// TIA Portal V18 export
// export: Created 2026-01-09T11:32:01.0889439Z, ExportSetting WithDefaults, DisplayName Totally Integrated Automation Portal, DisplayVersion V18 Update 5, DisplayName TIA Portal Openness, DisplayVersion V18 Update 5, DisplayName TIA Portal Teamcenter Gateway, DisplayVersion V18, DisplayName TIA Portal Version Control Interface, DisplayVersion V18, DisplayName SINAMICS Startdrive Advanced, DisplayVersion V18 SP2 Update 1, DisplayName SINAMICS Startdrive G110M, G120, G120C, G120D, G120P, G115D, DisplayVersion V18 SP2 Update 1, DisplayName SINAMICS Startdrive G130, G150, S120, S150, SINAMICS MV, S210, G220, S200, DisplayVersion V18 SP2 Update 1, DisplayName STEP 7 Professional, DisplayVersion V18 Update 5, DisplayName STEP 7 Safety, DisplayVersion V18, DisplayName WinCC Professional, DisplayVersion V18 Update 5
TagTable "Pilz"
  PilzData_85A1_I8 : Bool  (PLC tag PilzData.85A1.I8, CPU S71500-2PN_TP700, 100 ms)
  PilzData_85A1_I9 : Bool  (PLC tag PilzData.85A1.I9, CPU S71500-2PN_TP700, 100 ms)
  PilzData_85A1_I10 : Bool  (PLC tag PilzData.85A1.I10, CPU S71500-2PN_TP700, 100 ms)
  PilzData_85A1_I11 : Bool  (PLC tag PilzData.85A1.I11, CPU S71500-2PN_TP700, 100 ms)
  PilzData_85A1_I12 : Bool  (PLC tag PilzData.85A1.I12, CPU S71500-2PN_TP700, 100 ms)
  PilzData_85A1_I13 : Bool  (PLC tag PilzData.85A1.I13, CPU S71500-2PN_TP700, 100 ms)
  PilzData_85A1_I14 : Bool  (PLC tag PilzData.85A1.I14, CPU S71500-2PN_TP700, 100 ms)
  PilzData_85A1_I15 : Bool  (PLC tag PilzData.85A1.I15, CPU S71500-2PN_TP700, 100 ms)
  PilzData_85A1_I0 : Bool  (PLC tag PilzData.85A1.I0, CPU S71500-2PN_TP700, 100 ms)
  PilzData_85A1_I1 : Bool  (PLC tag PilzData.85A1.I1, CPU S71500-2PN_TP700, 100 ms)
  PilzData_85A1_I2 : Bool  (PLC tag PilzData.85A1.I2, CPU S71500-2PN_TP700, 100 ms)
  PilzData_85A1_I3 : Bool  (PLC tag PilzData.85A1.I3, CPU S71500-2PN_TP700, 100 ms)
  PilzData_85A1_I4 : Bool  (PLC tag PilzData.85A1.I4, CPU S71500-2PN_TP700, 100 ms)
  PilzData_85A1_I5 : Bool  (PLC tag PilzData.85A1.I5, CPU S71500-2PN_TP700, 100 ms)
  PilzData_85A1_I6 : Bool  (PLC tag PilzData.85A1.I6, CPU S71500-2PN_TP700, 100 ms)
  PilzData_85A1_I7 : Bool  (PLC tag PilzData.85A1.I7, CPU S71500-2PN_TP700, 100 ms)
  PilzData_85A1_I24 : Bool  (PLC tag PilzData.85A1.I24, CPU S71500-2PN_TP700, 100 ms)
  PilzData_85A1_I25 : Bool  (PLC tag PilzData.85A1.I25, CPU S71500-2PN_TP700, 100 ms)
  PilzData_85A1_I26 : Bool  (PLC tag PilzData.85A1.I26, CPU S71500-2PN_TP700, 100 ms)
  PilzData_85A1_I27 : Bool  (PLC tag PilzData.85A1.I27, CPU S71500-2PN_TP700, 100 ms)
  PilzData_85A1_I28 : Bool  (PLC tag PilzData.85A1.I28, CPU S71500-2PN_TP700, 100 ms)
  PilzData_85A1_I29 : Bool  (PLC tag PilzData.85A1.I29, CPU S71500-2PN_TP700, 100 ms)
  PilzData_85A1_I30 : Bool  (PLC tag PilzData.85A1.I30, CPU S71500-2PN_TP700, 100 ms)
  PilzData_85A1_I31 : Bool  (PLC tag PilzData.85A1.I31, CPU S71500-2PN_TP700, 100 ms)
  PilzData_85A1_I16 : Bool  (PLC tag PilzData.85A1.I16, CPU S71500-2PN_TP700, 100 ms)
  PilzData_85A1_I17 : Bool  (PLC tag PilzData.85A1.I17, CPU S71500-2PN_TP700, 100 ms)
  PilzData_85A1_I18 : Bool  (PLC tag PilzData.85A1.I18, CPU S71500-2PN_TP700, 100 ms)
  PilzData_85A1_I19 : Bool  (PLC tag PilzData.85A1.I19, CPU S71500-2PN_TP700, 100 ms)
  PilzData_85A1_I20 : Bool  (PLC tag PilzData.85A1.I20, CPU S71500-2PN_TP700, 100 ms)
  PilzData_85A1_I21 : Bool  (PLC tag PilzData.85A1.I21, CPU S71500-2PN_TP700, 100 ms)
  PilzData_85A1_I22 : Bool  (PLC tag PilzData.85A1.I22, CPU S71500-2PN_TP700, 100 ms)
  PilzData_85A1_I23 : Bool  (PLC tag PilzData.85A1.I23, CPU S71500-2PN_TP700, 100 ms)
  PilzData_85A1_O0 : Bool  (PLC tag PilzData.85A1.O0, CPU S71500-2PN_TP700, 100 ms)
  PilzData_85A1_O1 : Bool  (PLC tag PilzData.85A1.O1, CPU S71500-2PN_TP700, 100 ms)
  PilzData_85A1_O2 : Bool  (PLC tag PilzData.85A1.O2, CPU S71500-2PN_TP700, 100 ms)
  PilzData_85A1_O3 : Bool  (PLC tag PilzData.85A1.O3, CPU S71500-2PN_TP700, 100 ms)
  PilzData_85A1_Spare_1 : Bool  (PLC tag PilzData.85A1.Spare_1, CPU S71500-2PN_TP700, 100 ms)
  PilzData_85A1_Spare_2 : Bool  (PLC tag PilzData.85A1.Spare_2, CPU S71500-2PN_TP700, 100 ms)
  PilzData_85A1_Spare_3 : Bool  (PLC tag PilzData.85A1.Spare_3, CPU S71500-2PN_TP700, 100 ms)
  PilzData_85A1_Spare_4 : Bool  (PLC tag PilzData.85A1.Spare_4, CPU S71500-2PN_TP700, 100 ms)
  PilzData_85A1_Spare_5 : Bool  (PLC tag PilzData.85A1.Spare_5, CPU S71500-2PN_TP700, 100 ms)
  PilzData_85A1_Spare_6 : Bool  (PLC tag PilzData.85A1.Spare_6, CPU S71500-2PN_TP700, 100 ms)
  PilzData_85A1_Spare_7 : Bool  (PLC tag PilzData.85A1.Spare_7, CPU S71500-2PN_TP700, 100 ms)
  PilzData_85A1_Spare_8 : Bool  (PLC tag PilzData.85A1.Spare_8, CPU S71500-2PN_TP700, 100 ms)
  PilzData_85A1_Spare_9 : Bool  (PLC tag PilzData.85A1.Spare_9, CPU S71500-2PN_TP700, 100 ms)
  PilzData_85A1_Spare_10 : Bool  (PLC tag PilzData.85A1.Spare_10, CPU S71500-2PN_TP700, 100 ms)
  PilzData_85A1_Spare_11 : Bool  (PLC tag PilzData.85A1.Spare_11, CPU S71500-2PN_TP700, 100 ms)
  PilzData_85A1_Spare_12 : Bool  (PLC tag PilzData.85A1.Spare_12, CPU S71500-2PN_TP700, 100 ms)
  PilzData_85A2_I0 : Bool  (PLC tag PilzData.85A2.I0, CPU S71500-2PN_TP700, 100 ms)
  PilzData_85A2_I1 : Bool  (PLC tag PilzData.85A2.I1, CPU S71500-2PN_TP700, 100 ms)
  PilzData_85A2_I2 : Bool  (PLC tag PilzData.85A2.I2, CPU S71500-2PN_TP700, 100 ms)
  PilzData_85A2_I3 : Bool  (PLC tag PilzData.85A2.I3, CPU S71500-2PN_TP700, 100 ms)
  PilzData_85A2_I4 : Bool  (PLC tag PilzData.85A2.I4, CPU S71500-2PN_TP700, 100 ms)
  PilzData_85A2_I5 : Bool  (PLC tag PilzData.85A2.I5, CPU S71500-2PN_TP700, 100 ms)
  PilzData_85A2_I6 : Bool  (PLC tag PilzData.85A2.I6, CPU S71500-2PN_TP700, 100 ms)
  PilzData_85A2_I7 : Bool  (PLC tag PilzData.85A2.I7, CPU S71500-2PN_TP700, 100 ms)
  PilzData_85A2_O0 : Bool  (PLC tag PilzData.85A2.O0, CPU S71500-2PN_TP700, 100 ms)
  PilzData_85A2_O1 : Bool  (PLC tag PilzData.85A2.O1, CPU S71500-2PN_TP700, 100 ms)
  PilzData_85A2_O2 : Bool  (PLC tag PilzData.85A2.O2, CPU S71500-2PN_TP700, 100 ms)
  PilzData_85A2_O3 : Bool  (PLC tag PilzData.85A2.O3, CPU S71500-2PN_TP700, 100 ms)
  PilzData_85A2_Spare_1 : Bool  (PLC tag PilzData.85A2.Spare_1, CPU S71500-2PN_TP700, 100 ms)
  PilzData_85A2_Spare_2 : Bool  (PLC tag PilzData.85A2.Spare_2, CPU S71500-2PN_TP700, 100 ms)
  PilzData_85A2_Spare_3 : Bool  (PLC tag PilzData.85A2.Spare_3, CPU S71500-2PN_TP700, 100 ms)
  PilzData_85A2_Spare_4 : Bool  (PLC tag PilzData.85A2.Spare_4, CPU S71500-2PN_TP700, 100 ms)
  PilzData_85A3_I0 : Bool  (PLC tag PilzData.85A3.I0, CPU S71500-2PN_TP700, 100 ms)
  PilzData_85A3_I1 : Bool  (PLC tag PilzData.85A3.I1, CPU S71500-2PN_TP700, 100 ms)
  PilzData_85A3_I2 : Bool  (PLC tag PilzData.85A3.I2, CPU S71500-2PN_TP700, 100 ms)
  PilzData_85A3_I3 : Bool  (PLC tag PilzData.85A3.I3, CPU S71500-2PN_TP700, 100 ms)
  PilzData_85A3_I4 : Bool  (PLC tag PilzData.85A3.I4, CPU S71500-2PN_TP700, 100 ms)
  PilzData_85A3_I5 : Bool  (PLC tag PilzData.85A3.I5, CPU S71500-2PN_TP700, 100 ms)
  PilzData_85A3_I6 : Bool  (PLC tag PilzData.85A3.I6, CPU S71500-2PN_TP700, 100 ms)
  PilzData_85A3_I7 : Bool  (PLC tag PilzData.85A3.I7, CPU S71500-2PN_TP700, 100 ms)
  PilzData_85A3_O0 : Bool  (PLC tag PilzData.85A3.O0, CPU S71500-2PN_TP700, 100 ms)
  PilzData_85A3_O1 : Bool  (PLC tag PilzData.85A3.O1, CPU S71500-2PN_TP700, 100 ms)
  PilzData_85A3_O2 : Bool  (PLC tag PilzData.85A3.O2, CPU S71500-2PN_TP700, 100 ms)
  PilzData_85A3_O3 : Bool  (PLC tag PilzData.85A3.O3, CPU S71500-2PN_TP700, 100 ms)
  PilzData_85A3_Spare_1 : Bool  (PLC tag PilzData.85A3.Spare_1, CPU S71500-2PN_TP700, 100 ms)
  PilzData_85A3_Spare_2 : Bool  (PLC tag PilzData.85A3.Spare_2, CPU S71500-2PN_TP700, 100 ms)
  PilzData_85A3_Spare_3 : Bool  (PLC tag PilzData.85A3.Spare_3, CPU S71500-2PN_TP700, 100 ms)
  PilzData_85A3_Spare_4 : Bool  (PLC tag PilzData.85A3.Spare_4, CPU S71500-2PN_TP700, 100 ms)
  PilzData_Status : Int  (PLC tag PilzData.Status, CPU S71500-2PN_TP700, 100 ms)
  PilzData_85A4_I0 : Bool  (PLC tag PilzData.85A4.I0, CPU S71500-2PN_TP700, 100 ms)
  PilzData_85A4_I1 : Bool  (PLC tag PilzData.85A4.I1, CPU S71500-2PN_TP700, 100 ms)
  PilzData_85A4_I2 : Bool  (PLC tag PilzData.85A4.I2, CPU S71500-2PN_TP700, 100 ms)
  PilzData_85A4_I3 : Bool  (PLC tag PilzData.85A4.I3, CPU S71500-2PN_TP700, 100 ms)
  PilzData_85A4_I4 : Bool  (PLC tag PilzData.85A4.I4, CPU S71500-2PN_TP700, 100 ms)
  PilzData_85A4_I5 : Bool  (PLC tag PilzData.85A4.I5, CPU S71500-2PN_TP700, 100 ms)
  PilzData_85A4_I6 : Bool  (PLC tag PilzData.85A4.I6, CPU S71500-2PN_TP700, 100 ms)
  PilzData_85A4_I7 : Bool  (PLC tag PilzData.85A4.I7, CPU S71500-2PN_TP700, 100 ms)
  PilzData_85A4_O0 : Bool  (PLC tag PilzData.85A4.O0, CPU S71500-2PN_TP700, 100 ms)
  PilzData_85A4_O1 : Bool  (PLC tag PilzData.85A4.O1, CPU S71500-2PN_TP700, 100 ms)
  PilzData_85A4_O2 : Bool  (PLC tag PilzData.85A4.O2, CPU S71500-2PN_TP700, 100 ms)
  PilzData_85A4_O3 : Bool  (PLC tag PilzData.85A4.O3, CPU S71500-2PN_TP700, 100 ms)
  PilzData_85A4_Spare_1 : Bool  (PLC tag PilzData.85A4.Spare_1, CPU S71500-2PN_TP700, 100 ms)
  PilzData_85A4_Spare_2 : Bool  (PLC tag PilzData.85A4.Spare_2, CPU S71500-2PN_TP700, 100 ms)
  PilzData_85A4_Spare_3 : Bool  (PLC tag PilzData.85A4.Spare_3, CPU S71500-2PN_TP700, 100 ms)
  PilzData_85A4_Spare_4 : Bool  (PLC tag PilzData.85A4.Spare_4, CPU S71500-2PN_TP700, 100 ms)
  PilzData_85A5_I0 : Bool  (PLC tag PilzData.85A5.I0, CPU S71500-2PN_TP700, 100 ms)
  PilzData_85A5_I1 : Bool  (PLC tag PilzData.85A5.I1, CPU S71500-2PN_TP700, 100 ms)
  PilzData_85A5_I2 : Bool  (PLC tag PilzData.85A5.I2, CPU S71500-2PN_TP700, 100 ms)
  PilzData_85A5_I3 : Bool  (PLC tag PilzData.85A5.I3, CPU S71500-2PN_TP700, 100 ms)
  PilzData_85A5_I4 : Bool  (PLC tag PilzData.85A5.I4, CPU S71500-2PN_TP700, 100 ms)
  PilzData_85A5_I5 : Bool  (PLC tag PilzData.85A5.I5, CPU S71500-2PN_TP700, 100 ms)
  PilzData_85A5_I6 : Bool  (PLC tag PilzData.85A5.I6, CPU S71500-2PN_TP700, 100 ms)
  PilzData_85A5_I7 : Bool  (PLC tag PilzData.85A5.I7, CPU S71500-2PN_TP700, 100 ms)
  PilzData_85A5_O0 : Bool  (PLC tag PilzData.85A5.O0, CPU S71500-2PN_TP700, 100 ms)
  PilzData_85A5_O1 : Bool  (PLC tag PilzData.85A5.O1, CPU S71500-2PN_TP700, 100 ms)
  PilzData_85A5_O2 : Bool  (PLC tag PilzData.85A5.O2, CPU S71500-2PN_TP700, 100 ms)
  PilzData_85A5_O3 : Bool  (PLC tag PilzData.85A5.O3, CPU S71500-2PN_TP700, 100 ms)
  PilzData_85A5_Spare_1 : Bool  (PLC tag PilzData.85A5.Spare_1, CPU S71500-2PN_TP700, 100 ms)
  PilzData_85A5_Spare_2 : Bool  (PLC tag PilzData.85A5.Spare_2, CPU S71500-2PN_TP700, 100 ms)
  PilzData_85A5_Spare_3 : Bool  (PLC tag PilzData.85A5.Spare_3, CPU S71500-2PN_TP700, 100 ms)
  PilzData_85A5_Spare_4 : Bool  (PLC tag PilzData.85A5.Spare_4, CPU S71500-2PN_TP700, 100 ms)
